// TIA Portal project "teste_variaveis_09_02" (V17)
// HARDWARE PADRAO CLP, INTERFACES E IHM

(* hardware
DEVICE "S7-1500/ET200MP station_1"  S7-1500 station
   slot 0: "Rail_0"  Rack  6ES7 590-1***0-0AA0
   slot 1: "PLC_1"  CPU 1516-3 PN/DP  6ES7 516-3AN01-0AB0  V2.9
      slot 3: "CPU display_1"  6ES7591-1BA00-0AA0
      slot 32768: "PROFINET interface_1"  X1
      slot 33024: "PROFINET interface_2"  X2
      slot 33280: "DP interface_1"  X3
      slot 34817: "Virtual CP interface port_1"  Virtual CP interface port  Virtual CP interface port
   slot 2: "DI 32x24VDC HF_1"  DI 32x24VDC HF  6ES7 521-1BL00-0AB0  V2.1
   slot 3: "DQ 32x24VDC/0.5A HF_1"  DQ 32x24VDC/0.5A HF  6ES7 522-1BL01-0AB0  V1.0
   slot 4: "AI 8xU/I/RTD/TC ST_1"  AI 8xU/I/RTD/TC ST  6ES7 531-7KF00-0AB0  V2.0
   slot 5: "AQ 4xU/I ST_1"  AQ 4xU/I ST  6ES7 532-5HD00-0AB0  V2.0
DEVICE "HMI_1"  KTP700 Basic PN
   slot 0: "HMI_1"  KTP700 Basic PN  6AV2 123-2GB03-0AX0  14.0.1.0
   slot 1: "HMI_RT_1"  KTP700 Basic PN  6AV2 123-2GB03-0AX0  14.0.1.0
   slot 5: "HMI_1.IE_CP_1"  PROFINET Interface  14.0.1.0
      slot 1: "PROFINET Interface_1"  PROFINET Interface
         slot 1: "Port_1"  Port
*)

// ===== PLC "PLC_1"  CPU 1516-3 PN/DP =====

VAR_GLOBAL   // PLC tag table "Default tag table"
   "Clock_Byte" AT %MB100 : Byte;
   "Clock_10Hz" AT %M100.0 : Bool;
   "Clock_5Hz" AT %M100.1 : Bool;
   "Clock_2.5Hz" AT %M100.2 : Bool;
   "Clock_2Hz" AT %M100.3 : Bool;
   "Clock_1.25Hz" AT %M100.4 : Bool;
   "Clock_1Hz" AT %M100.5 : Bool;
   "Clock_0.625Hz" AT %M100.6 : Bool;
   "Clock_0.5Hz" AT %M100.7 : Bool;
END_VAR

VAR_GLOBAL   // PLC tag table "entradas_fisicas"
   "on" AT %I1.1 : Bool;
   "off" AT %I1.2 : Bool;
   "canal_0_300" AT %IW6 : Int;
   "eme" AT %I1.3 : Bool;
END_VAR

VAR_GLOBAL   // PLC tag table "saidas_fisicas"
   "sinVD" AT %Q1.1 : Bool;
   "sinVM" AT %Q1.3 : Bool;
   "canal_0_400" AT %QW4 : Int;
END_VAR

DATA_BLOCK "Data_block_1"   // DB1
{ S7_Optimized_Access := 'TRUE' }
VERSION : 0.1
   VAR
      status : String;
      tensaoMedida_300 : Real;
      tensaoDesejada_400 : Real;
      ihmOn : Bool;
      ihmOff : Bool;
      leitura_300 : Real;
      escrita_400 : Real;
      trocarTelas : Array[0..3] of Int;
      scanEme : Bool;
   END_VAR
BEGIN
END_DATA_BLOCK

FUNCTION "trocarTelas" : Void   // FC1, LAD
{ S7_Optimized_Access := 'TRUE' }
VERSION : 0.1
   VAR_TEMP   // added for the SCL form of the ladder/FBD networks
      _w1 : Bool;
   END_VAR
BEGIN

REGION Network 1: COMANDO PRA TOCAR TELA QUANDO A EMERGÊNCIA
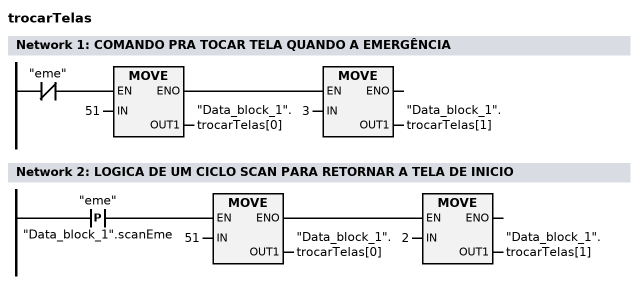
   RUNG wire#powerrail
      I_Contact( "eme" )
      Move(in := 51, out1 => "Data_block_1".trocarTelas[0])
      Move(in := 3, out1 => "Data_block_1".trocarTelas[1])
   END_RUNG
   // the same network as SCL:
   IF NOT "eme" THEN
       "Data_block_1".trocarTelas[0] := 51;
       "Data_block_1".trocarTelas[1] := 3;
   END_IF;
END_REGION

REGION Network 2: LOGICA DE UM CICLO SCAN PARA RETORNAR A TELA DE INICIO
   RUNG wire#powerrail
      P_Contact(operand := "eme", bit := "Data_block_1".scanEme)
      Move(in := 51, out1 => "Data_block_1".trocarTelas[0])
      Move(in := 2, out1 => "Data_block_1".trocarTelas[1])
   END_RUNG
   // the same network as SCL:
   #_w1 := "eme" AND NOT "Data_block_1".scanEme;   // rising edge of "eme"
   "Data_block_1".scanEme := "eme";
   IF #_w1 THEN
       "Data_block_1".trocarTelas[0] := 51;
       "Data_block_1".trocarTelas[1] := 2;
   END_IF;
END_REGION
END_FUNCTION

ORGANIZATION_BLOCK "Main"   // OB1, LAD, ProgramCycle
TITLE = "Main Program Sweep (Cycle)"
{ S7_Optimized_Access := 'TRUE' }
VERSION : 0.1
   VAR_INPUT
      Initial_Call : Bool;   // Initial call of this OB
      Remanence : Bool;   // =True, if remanent data are available
   END_VAR
BEGIN

REGION Network 1
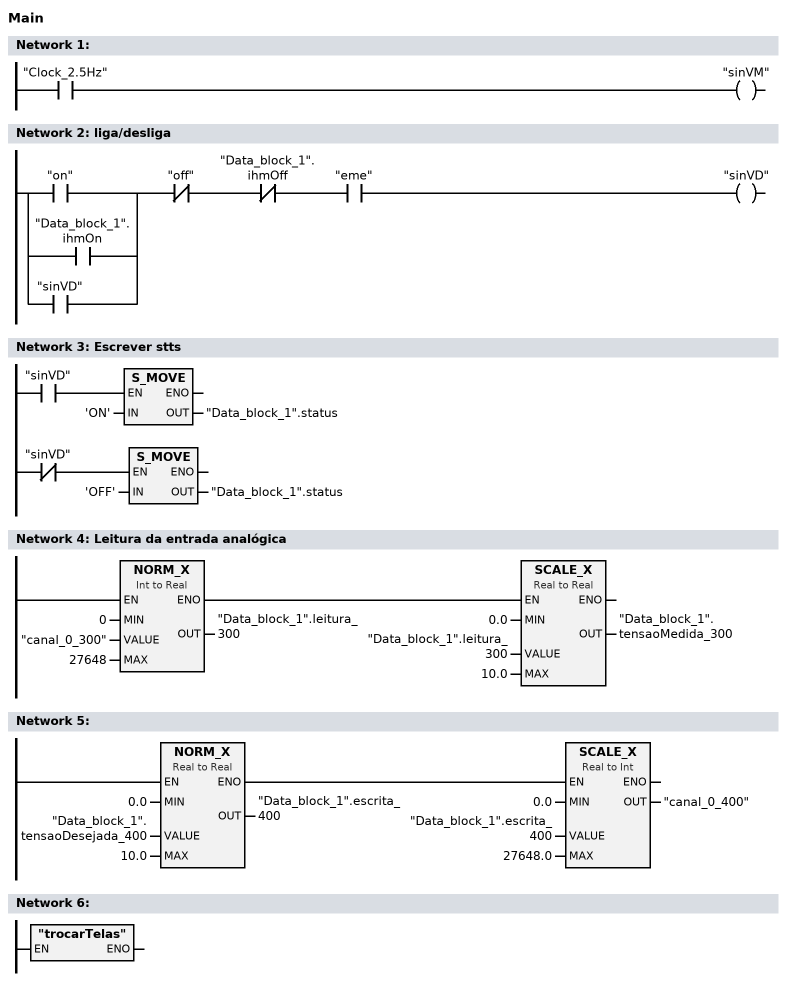
   RUNG wire#powerrail
      Contact( "Clock_2.5Hz" )
      Coil( "sinVM" )
   END_RUNG
   // the same network as SCL:
   "sinVM" := "Clock_2.5Hz";
END_REGION

REGION Network 2: liga/desliga
   RUNG wire#powerrail
      Contact( "on" )
      wire#w1
      I_Contact( "off" )
      I_Contact( "Data_block_1".ihmOff )
      Contact( "eme" )
      Coil( "sinVD" )
   END_RUNG
   RUNG wire#powerrail
      Contact( "Data_block_1".ihmOn )
   END_RUNG wire#w1
   RUNG wire#powerrail
      Contact( "sinVD" )
   END_RUNG wire#w1
   // the same network as SCL:
   "sinVD" := ("on" OR "Data_block_1".ihmOn OR "sinVD") AND NOT "off" AND NOT "Data_block_1".ihmOff AND "eme";
END_REGION

REGION Network 3: Escrever stts
   RUNG wire#powerrail
      Contact( "sinVD" )
      S_Move(in := 'ON', out => "Data_block_1".status)
   END_RUNG
   RUNG wire#powerrail
      I_Contact( "sinVD" )
      S_Move(in := 'OFF', out => "Data_block_1".status)
   END_RUNG
   // the same network as SCL:
   IF "sinVD" THEN "Data_block_1".status := 'ON'; END_IF;
   IF NOT "sinVD" THEN "Data_block_1".status := 'OFF'; END_IF;
END_REGION

REGION Network 4: Leitura da entrada analógica
   RUNG wire#powerrail
      { S7_Templates := "[SrcType := Int, DestType := Real]" } Normalize(min := 0, value := "canal_0_300", max := 27648, out => "Data_block_1".leitura_300)
      { S7_Templates := "[SrcType := Real, DestType := Real]" } Scale(min := 0.0, value := "Data_block_1".leitura_300, max := 10.0, out => "Data_block_1".tensaoMedida_300)
   END_RUNG
   // the same network as SCL:
   "Data_block_1".leitura_300 := NORM_X(MIN := 0, VALUE := "canal_0_300", MAX := 27648);
   "Data_block_1".tensaoMedida_300 := SCALE_X(MIN := 0.0, VALUE := "Data_block_1".leitura_300, MAX := 10.0);
END_REGION

REGION Network 5
   RUNG wire#powerrail
      { S7_Templates := "[SrcType := Real, DestType := Real]" } Normalize(min := 0.0, value := "Data_block_1".tensaoDesejada_400, max := 10.0, out => "Data_block_1".escrita_400)
      { S7_Templates := "[SrcType := Real, DestType := Int]" } Scale(min := 0.0, value := "Data_block_1".escrita_400, max := 27648.0, out => "canal_0_400")
   END_RUNG
   // the same network as SCL:
   "Data_block_1".escrita_400 := NORM_X(MIN := 0.0, VALUE := "Data_block_1".tensaoDesejada_400, MAX := 10.0);
   "canal_0_400" := SCALE_X(MIN := 0.0, VALUE := "Data_block_1".escrita_400, MAX := 27648.0);
END_REGION

REGION Network 6
   RUNG wire#powerrail
      "trocarTelas"()
   END_RUNG
   // the same network as SCL:
   "trocarTelas"();
END_REGION
END_ORGANIZATION_BLOCK

(* ===== HMI "HMI_RT_1" =====
system functions are stored by id; their names below are inferred from use
connection "HMI_Connection_1": ETHERNET, SMART_S7_1500_OMS

HMI tags "Default tag table"
   "sinVM" : Bool = PLC sinVM AT %Q1.3, 1 s
   "sinVD" : Bool = PLC sinVD AT %Q1.1, 1 s
   "Data_block_1_ihmOn" : Bool = PLC Data_block_1.ihmOn, 1 s
   "Data_block_1_ihmOff" : Bool = PLC Data_block_1.ihmOff, 1 s
   "Data_block_1_status" : String[254] = PLC Data_block_1.status, 1 s
   "Data_block_1_tensaoDesejada_400" : Real = PLC Data_block_1.tensaoDesejada_400, 1 s
   "Data_block_1_tensaoMedida_300" : Real = PLC Data_block_1.tensaoMedida_300, 1 s

text list "volt": 0 '0V'; 2 '2V'; 4 '4V'; 6 '6V'; 8 '8V'; 10 '10V'

Template "Template_1" 800x480
   Button "Exit" at 714,429 size 71x50; TextOff 'Exit'; PictureOff "ExitRuntime_KTP700_Basic_PN_TR"; PictureOn "ExitRuntime_KTP700_Basic_PN_TR"
      on Release: StopRuntime(0)
   Button "Template_Button" at 614,429 size 71x50; TextOff 'Text'
   Button "Template_Button_1" at 514,429 size 71x50; TextOff 'Text'
   Button "Template_Button_2" at 414,429 size 71x50; TextOff 'Text'
   Button "Template_Button_3" at 314,429 size 71x50; TextOff 'Text'
   Button "Template_Button_4" at 214,429 size 71x50; TextOff 'Text'
   Button "Template_Button_5" at 114,429 size 71x50; TextOff 'Text'
   Button "Start screen" at 14,429 size 71x50; TextOff 'Start screen'; PictureOff "NavigateHome_KTP700_Basic_PN_TR"; PictureOn "NavigateHome_KTP700_Basic_PN_TR"
      on Release: ActivateScreen("Root screen", 0)

screen "Root screen" 800x480, template "Template_1"
   Softkey "Softkey_F2" at 0,0 size 0x0; SoftkeyImage "Left_Arrow"
      on KeyDown: ActivateScreen("INICIO", 2)
   TextField "Text field_1" at 308,16 size 191x33; Text 'PROJETO TESTE'
   TextField "Text field_2" at 64,37 size 121x27; Text 'OSCILADOR'
   Circle "Circle_1" at 86,63 size 76x76
      Appearance <- "sinVM"
   Circle "Circle_2" at 279,113 size 27x27
      Appearance <- "sinVM"
   Circle "Circle_3" at 514,114 size 27x27
      Appearance <- "sinVM"
   TextField "Text field_3" at 120,155 size 95x27; Text 'ON / OFF'
   Circle "Circle_4" at 179,184 size 76x76
      Appearance <- "sinVD"
   Button "Button_1" at 411,150 size 110x49; TextOff 'ON'
      on Press: function_b14e0dd5("Data_block_1_ihmOn", 0)
      Visibility <- "sinVD"
   Button "Button_2" at 491,174 size 109x49; TextOff 'OFF'
      on Press: function_b14e0dd5("Data_block_1_ihmOff", 0)
      Visibility <- "sinVD"
   IOField "I/O field_1" at 10,4 size 234x32; FormatPattern ?????
      ProcessValue <- "Data_block_1_status"
   TextField "Text field_4" at 638,9 size 96x23; Text 'VOLTAGEM'
   IOField "I/O field_2" at 672,107 size 121x32; FormatPattern 99.99; Unit V
      ProcessValue <- "Data_block_1_tensaoMedida_300"
   TextField "Text field_5" at 562,54 size 101x23; Text 'Injeção 400'
   SymbolicIOField "Symbolic I/O field_1" at 672,50 size 121x33; TextOff '0'; TextOn '1'; TextList "volt"
      ProcessValue <- "Data_block_1_tensaoDesejada_400"
   TextField "Text field_6" at 562,111 size 107x23; Text 'Medição 300'
   TextField "Text field_7" at 16,8 size 69x22; Text 'STATUS:'
   Bar "Bar_1" at 670,152 size 123x202; MinimumValue 0; MaximumValue 10
      ProcessValue <- "Data_block_1_tensaoMedida_300"
   TrendView "Trend view_1" at 9,265 size 233x154

screen "INICIO" 800x480
   GraphicView "Graphic view_1" at 0,0 size 800x479; Picture "coriga1"
   GraphicView "Graphic view_2" at 229,126 size 105x37; Picture "coriga1"
   GraphicView "Graphic view_3" at 471,123 size 105x37; Picture "coriga1"
   Softkey "Softkey_F3" at 0,0 size 0x0; SoftkeyImage "Right_Arrow"
      on KeyDown: ActivateScreen("Root screen", 1)

screen "Tela_emergencia" 800x480
   GraphicView "Graphic view_1" at 0,0 size 799x479; Picture "BATAM"
   TextField "Text field_1" at 199,75 size 394x34; Text 'EITA BIXO EMERGÊNCIA kkkkk'
*)